FUNCTION_BLOCK fbMotorHomingAxis
VAR_INPUT

	bEmergencyButton: BOOL;
	bHomingStart : BOOL ;
	lMoveVelo : LREAL;
	lMoveAcc : LREAL;
	lMoveDcc : LREAL;
	lMove2ndVelo : LREAL;
	lMove2ndAcc : LREAL;
	lMove2ndDcc : LREAL;
	bHomeSensor1 : BOOL;
	bOverTravelSensor1 : BOOL;
	bOverTravelSensor2 : BOOL;
	bReset : BOOL;
	tAlwaysHomeCompleteTimeDelay: TIME;
	tMCHomeStartDelay: TIME;


END_VAR

VAR_IN_OUT
	Axis1	: Axis_Ref;
	lrCurrentAxisPos : LREAL;
END_VAR

VAR_OUTPUT

	Home1Complete : BOOL;
END_VAR
VAR

	lrPosAxisAwayHome : LREAL := 9999;

	ArmStopBit: BOOL;
	HomingInterlocking: BOOL;
	ArmTouchHome: BOOL;
	bOverTravelSensor: BOOL;
	halt: MC_Halt;
	ArmHaltDone: BOOL;
	ArmBelowSensor: BOOL;
	bHomeSensor: BOOL;
	Move2home: BOOL;
	move1: MC_MoveRelative;
	moveBusy: BOOL;
	halt1: MC_Halt;
	ArmEstopDone: BOOL;
	Estop: BOOL;
	MoveAway: BOOL;
	move2: MC_MoveRelative;
	Timer1: TON;
	ArmAwayHome: BOOL;
	move3: MC_MoveRelative;
	AwayHomeBusy: BOOL;
	AwayHomeDone: BOOL;
	halt3: MC_Halt;
	AwayHaltDone: BOOL;
	HomingStart: BOOL;
	Delay: TON;
	Timer2: TON;
	home1: MC_Home;
	Home1Done: BOOL;
	Timer3: TON;
	step1: BOOL;
	Delay1: TON;
	HomeStartDIFU: R_TRIG;
	bPosError: BOOL;
	MCSP: MC_SetPosition;
	HomingStartEN_DIFU: R_TRIG;
	HomingStartFE: F_TRIG;
	PosErrorDIFU: R_TRIG;
	PosErrorTimer: TON;
	Home1Complete1: BOOL;
	Home1CompleteDIFU: R_TRIG;
	DON: TON;
END_VAR

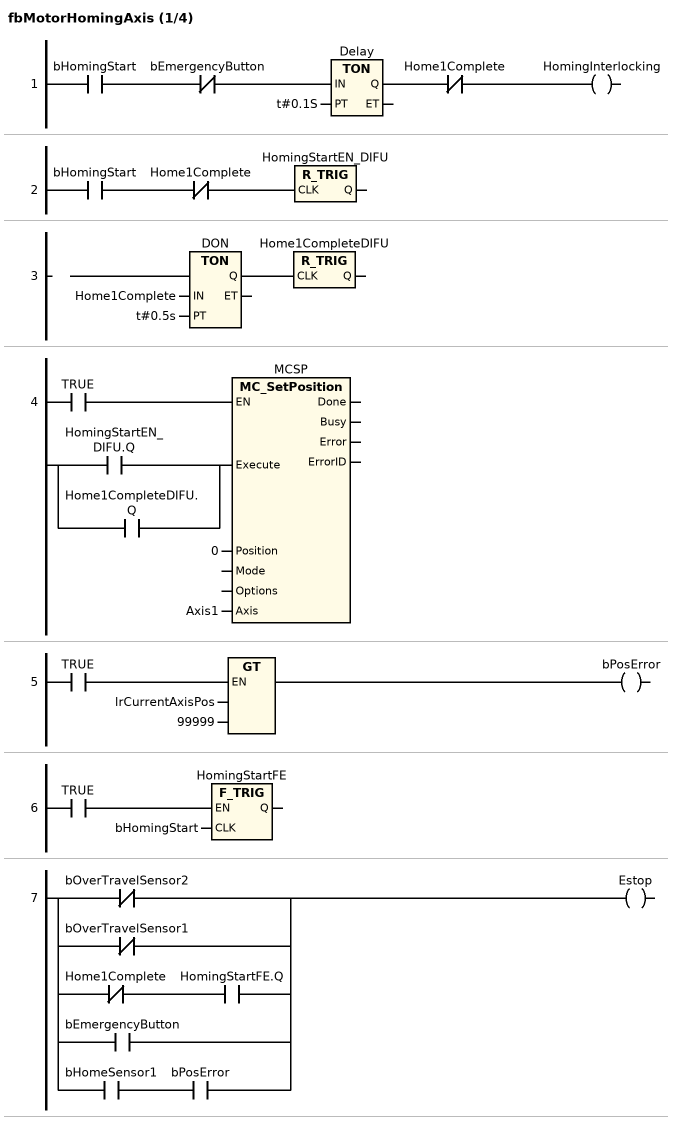
// NETWORK 1
Delay(IN := bHomingStart AND NOT bEmergencyButton, PT := t#0.1S); // TON
HomingInterlocking := Delay.Q AND NOT Home1Complete;

// NETWORK 2
HomingStartEN_DIFU(CLK := bHomingStart AND NOT Home1Complete); // R_TRIG

// NETWORK 3
DON(IN := Home1Complete, PT := t#0.5s); // TON
Home1CompleteDIFU(CLK := DON.Q); // R_TRIG

// NETWORK 4
MCSP(Execute := HomingStartEN_DIFU.Q OR Home1CompleteDIFU.Q, Position := 0, Axis := Axis1); // MC_SetPosition

// NETWORK 5
bPosError := lrCurrentAxisPos > 99999;

// NETWORK 6
HomingStartFE(CLK := bHomingStart); // F_TRIG

// NETWORK 7
Estop := NOT bOverTravelSensor2 OR NOT bOverTravelSensor1 OR NOT Home1Complete AND HomingStartFE.Q OR bEmergencyButton OR bHomeSensor1 AND bPosError;

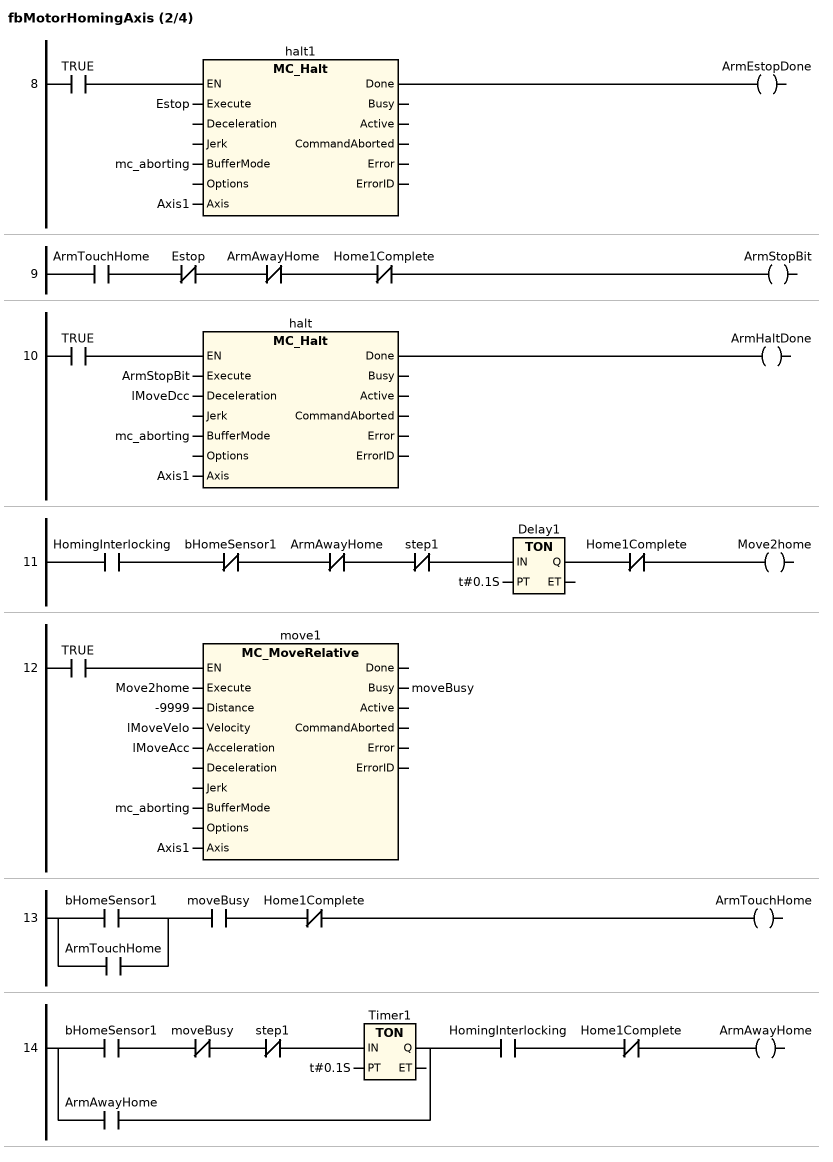
// NETWORK 8
halt1(Execute := Estop, BufferMode := mc_aborting, Axis := Axis1); // MC_Halt
ArmEstopDone := halt1.Done;

// NETWORK 9
ArmStopBit := ArmTouchHome AND NOT Estop AND NOT ArmAwayHome AND NOT Home1Complete;

// NETWORK 10
halt(Execute := ArmStopBit, Deceleration := lMoveDcc, BufferMode := mc_aborting, Axis := Axis1); // MC_Halt
ArmHaltDone := halt.Done;

// NETWORK 11
Delay1(IN := HomingInterlocking AND NOT bHomeSensor1 AND NOT ArmAwayHome AND NOT step1, PT := t#0.1S); // TON
Move2home := Delay1.Q AND NOT Home1Complete;

// NETWORK 12
move1(
    Execute := Move2home,
    Distance := -9999,
    Velocity := lMoveVelo,
    Acceleration := lMoveAcc,
    BufferMode := mc_aborting,
    Axis := Axis1,
    Busy => moveBusy); // MC_MoveRelative

// NETWORK 13
ArmTouchHome := (bHomeSensor1 OR ArmTouchHome) AND moveBusy AND NOT Home1Complete;

// NETWORK 14
Timer1(IN := bHomeSensor1 AND NOT moveBusy AND NOT step1, PT := t#0.1S); // TON
ArmAwayHome := (Timer1.Q OR ArmAwayHome) AND HomingInterlocking AND NOT Home1Complete;

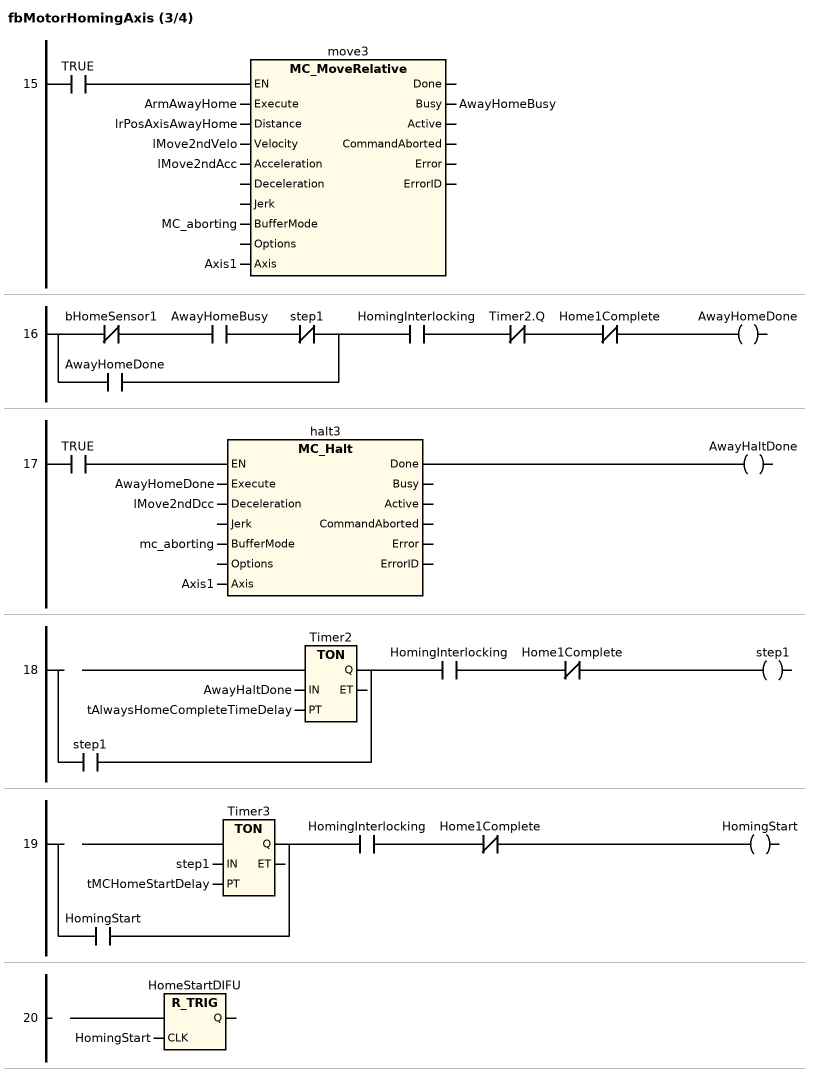
// NETWORK 15
move3(
    Execute := ArmAwayHome,
    Distance := lrPosAxisAwayHome,
    Velocity := lMove2ndVelo,
    Acceleration := lMove2ndAcc,
    BufferMode := MC_aborting,
    Axis := Axis1,
    Busy => AwayHomeBusy); // MC_MoveRelative

// NETWORK 16
AwayHomeDone := (NOT bHomeSensor1 AND AwayHomeBusy AND NOT step1 OR AwayHomeDone) AND HomingInterlocking AND NOT Timer2.Q AND NOT Home1Complete;

// NETWORK 17
halt3(Execute := AwayHomeDone, Deceleration := lMove2ndDcc, BufferMode := mc_aborting, Axis := Axis1); // MC_Halt
AwayHaltDone := halt3.Done;

// NETWORK 18
Timer2(IN := AwayHaltDone, PT := tAlwaysHomeCompleteTimeDelay); // TON
step1 := (Timer2.Q OR step1) AND HomingInterlocking AND NOT Home1Complete;

// NETWORK 19
Timer3(IN := step1, PT := tMCHomeStartDelay); // TON
HomingStart := (Timer3.Q OR HomingStart) AND HomingInterlocking AND NOT Home1Complete;

// NETWORK 20
HomeStartDIFU(CLK := HomingStart); // R_TRIG

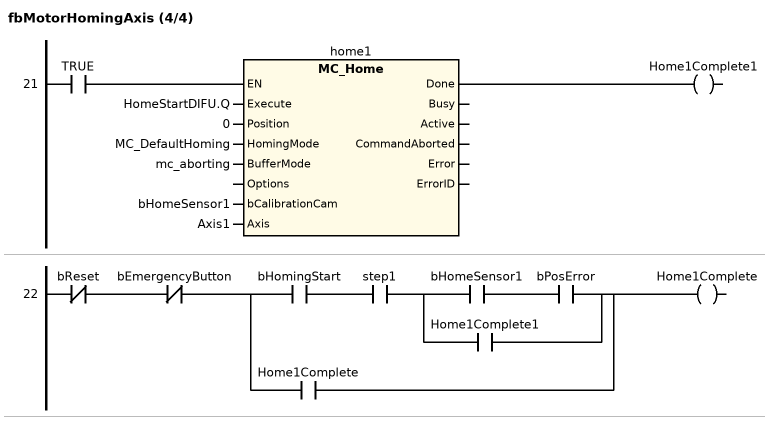
// NETWORK 21
home1(
    Execute := HomeStartDIFU.Q,
    Position := 0,
    HomingMode := MC_DefaultHoming,
    BufferMode := mc_aborting,
    bCalibrationCam := bHomeSensor1,
    Axis := Axis1); // MC_Home
Home1Complete1 := home1.Done;

// NETWORK 22
Home1Complete := NOT bReset AND NOT bEmergencyButton AND (bHomingStart AND step1 AND (bHomeSensor1 AND bPosError OR Home1Complete1) OR Home1Complete);

END_FUNCTION_BLOCK

(* stored: Version 1.1.0.1, ProductVersion 3.1.4024.12
   POU fbMotorHomingAxis: Id {814edeac-47e6-4bbe-b83c-c3657d13f5af}, SpecialFunc None *)
